(* PLC project Generated.project, CODESYS CODESYS V3.5 SP19 Patch 1 *)
(* stored: creationDateTime 2026-09-23T12:01:01.984454, modificationDateTime 2026-09-23T12:01:01.984454 *)

(* ═══════════════════════════════════════════════════════════════ ST_TranslationCfg — Configurations et paramètres réglables pour Translation M3 ─────────────────────────────────────────────────────────────── 🎨 Destiné au paramétrage depuis l'IHM (RETAIN) — même patron que ST_WinchCfg. 📄 Vitesses de ralentissement d'approche réglables depuis l'IHM (RETAIN), même patron que ST_WinchCfg. ═══════════════════════════════════════════════════════════════ *)
TYPE ST_TranslationCfg : STRUCT
  CfgApproachSpeedTremie_Hz : REAL := 20;  (* 🐢 Vitesse réduite d'approche Trémie (Hz), déclenchée par capteur PV, Direction=1 — reglage nominal confirme operateur *)
  CfgApproachSpeedMaintenance_Hz : REAL := 20;  (* 🐢 Vitesse réduite d'approche Maintenance (Hz), déclenchée par capteur P1, Direction=-1 — reglage nominal confirme operateur *)
  CfgApproachSpeedP1_Hz : REAL := 20;  (* 🐢 Vitesse réduite d'approche P1 (Hz), déclenchée par capteur P2, Direction=-1 — reglage nominal confirme operateur *)
  Initialized : BOOL := FALSE;  (* Flag restauration boot (défaut FALSE non ambigu) — même patron que ST_WinchCfg 🚦 TRUE = config restaurée depuis GVL_PERSISTENT ce boot *)
END_STRUCT;
END_TYPE
